Omron Sysmac Studio project Function blocks Multiaxis library (Sysmac Studio 1.56.0.64011, StandardProject)

# Controller new_Controller_0: NJ301-1200 version 1.64
Units and slaves: Alimentación : NJ-Px3001; CPU : NJ301-1200

FUNCTION_BLOCK PowerAxes
(* Libreria de ejes *)
VAR
    PowerAxis : MC_Power;
    PosAxis : INT;
    DataAxes : ARRAY[0..50] OF _sAXIS_REF;
    DataPos : INT;
END_VAR
VAR_IN_OUT
    InputAxes : ARRAY[0..50] OF _sAXIS_REF;
    AxisNumbers : INT;
END_VAR
VAR_INPUT
    InputPowerEnable : ARRAY[0..50] OF bool;
END_VAR
VAR_OUTPUT
    OutPowerStatus : ARRAY[0..50] OF bool;
    OutPowerBusy : ARRAY[0..50] OF bool;
    OutPowerError : ARRAY[0..50] OF bool;
    OutPowerErrorID : ARRAY[0..50] OF word;
    DataPositionOut : INT;
    DataAxesOut : ARRAY[0..50] OF _sAXIS_REF;
END_VAR
(*************************************************************************************************************
                                        Function block: Axes block programming
**************************************************************************************************************

*    Project: CNC Machine
*    Equipment: Omron NJ301-1200 PLC
*    Description: Axes power parameter setting function
*    Date: 23/06/2024

**************************************************************************************************************)

// This is the main function of the library:
// The operation of the whole library relies on arrays of [0..50] so the max limit of servos would be 50.
// It records the total number of servo axes and performs the PowerAxis function to power the servos.
// AxisNumbers - input variable for comparison. The total number of servo axes is stored in this variable.
// PosAxis - counter variable. It is in charge of counting and adding up to the indicated value.
// DataPositionOut - counter output variable that is responsible for traversing the main data structure in the main.
// InputAxes - input array variable _sAXIS_REF, which corresponds to servo system variables.
// DataAxesOut - output array variable _sAXIS_REF, this variable outputs the servo axes status information.
// PowerAxis - Motion Control function corresponding to MC_Power.

PosAxis:= PosAxis+1;

IF PosAxis >=AxisNumbers THEN
	PosAxis:= 0;
END_IF;

DataPos:= PosAxis;

(***********  Asignation of data estructure  ***********)

// Inputs
DataAxes[DataPos]:= InputAxes[DataPos];

// Outputs
DataPositionOut:= DataPos;
DataAxesOut[DataPos]:= DataAxes[DataPos];

(*  ENABLE MACHINE AXES POWER  *)

PowerAxis(Axis:=InputAxes[DataPos], Enable:=InputPowerEnable[DataPos], Status=>OutPowerStatus[DataPos], 
			Busy=>OutPowerBusy[DataPos], Error=>OutPowerError[DataPos], ErrorID=>OutPowerErrorID[DataPos]);

// BLOCK END
END_FUNCTION_BLOCK

FUNCTION_BLOCK HomingAxes
(* Libreria de ejes *)
VAR
    OriginAxis : MC_Home;
    DataPos : INT;
END_VAR
VAR_IN_OUT
    InputAxes : ARRAY[0..50] OF _sAXIS_REF;
    InputDataPosition : INT;
END_VAR
VAR_INPUT
    InputOrginExecute : ARRAY[0..50] OF bool;
END_VAR
VAR_OUTPUT
    OutOriginDone : ARRAY[0..50] OF bool;
    OutOriginBusy : ARRAY[0..50] OF bool;
    OutOriginAborted : ARRAY[0..50] OF bool;
    OutOriginError : ARRAY[0..50] OF bool;
    OutOriginErrorID : ARRAY[0..50] OF word;
END_VAR
(*************************************************************************************************************
                                        Function block: Axes block programming
**************************************************************************************************************

*    Project: CNC Machine
*    Equipment: Omron NJ301-1200 PLC
*    Description: Axes parameter origin function
*    Date: 23/06/2024

**************************************************************************************************************)

// This is the Homing function of the library:
// The operation of the whole library relies on arrays of [0..50] so the max limit of servos would be 50.
// Performs the origin positioning of the servo axes.
// InputDataPosition - input variable in which is indicated to which servo axis should make the homing reference.
// InputAxes - input array variable _sAXIS_REF, which corresponds to servo system variables.
// OriginAxis - Motion Control function corresponding to MC_Home.

DataPos:= InputDataPosition;

(*  ENABLE MACHINE AXES HOMING  *)

OriginAxis(Axis:=InputAxes[DataPos], Execute:=InputOrginExecute[DataPos], Done=>OutOriginDone[DataPos], Busy=>OutOriginBusy[DataPos],
			 CommandAborted=>OutOriginAborted[DataPos], Error=>OutOriginError[DataPos], ErrorID=>OutOriginErrorID[DataPos]);

// BLOCK END
END_FUNCTION_BLOCK

FUNCTION_BLOCK JogAxes
(* Libreria de ejes *)
VAR
    JogAxis : MC_MoveJog;
    DataPos : INT;
END_VAR
VAR_IN_OUT
    InputAxes : ARRAY[0..50] OF _sAXIS_REF;
END_VAR
VAR_INPUT
    InputDataPosition : INT;
    InputJogPositive : ARRAY[0..50] OF bool;
    InputJogNegative : ARRAY[0..50] OF bool;
    InputJogVelocity : ARRAY[0..50] OF lreal;
    InputJogAcceleration : ARRAY[0..50] OF lreal;
    InputJogDeceleration : ARRAY[0..50] OF lreal;
END_VAR
VAR_OUTPUT
    OutJogBusy : ARRAY[0..50] OF bool;
    OutJogAborted : ARRAY[0..50] OF bool;
    OutJogError : ARRAY[0..50] OF bool;
    OutJogErrorID : ARRAY[0..50] OF word;
END_VAR
(*************************************************************************************************************
                                        Function block: Axes block programming
**************************************************************************************************************

*    Project: CNC Machine
*    Equipment: Omron NJ301-1200 PLC
*    Description: Axes parameter jog function
*    Date: 23/06/2024

**************************************************************************************************************)

// This is the Jog function of the library:
// The operation of the whole library relies on arrays of [0..50] so the max limit of servos would be 50.
// Performs the free Jog movement of the servo axes.
// InputDataPosition - input variable in which is indicated to which servo axis should make the homing reference.
// InputAxes - input array variable _sAXIS_REF, which corresponds to servo system variables.
// JogAxis - Motion Control function corresponding to MC_MoveJog.

DataPos:= InputDataPosition;

(*  ENABLE MACHINE AXES JOG  *)

JogAxis(Axis:=InputAxes[DataPos], PositiveEnable:=InputJogPositive[DataPos], NegativeEnable:=InputJogNegative[DataPos],
		Velocity:=InputJogVelocity[DataPos], Acceleration:=InputJogAcceleration[DataPos], Deceleration:=InputJogDeceleration[DataPos],
		Busy=>OutJogBusy[DataPos], CommandAborted=>OutJogAborted[DataPos], Error=>OutJogError[DataPos], ErrorID=>OutJogErrorID[DataPos]);

// BLOCK END
END_FUNCTION_BLOCK